FUNCTION_BLOCK LIGHTS_CYCLE (* Composite Function Block Type *)
  (* Standard: 61499-2 *)
  (* Version 0.2, 2003-12-05, JHC, Rockwell Automation, Renamed from NEWCOMPFB. *)
  (* Version 0.1, 2002-01-08, JHC, Rockwell Automation, Added DLY FB as example. *)
  (* Version 0.0, 2000-05-27, JHC, Rockwell Automation *)
  (* Compiler header: package fb.rt.student; *)
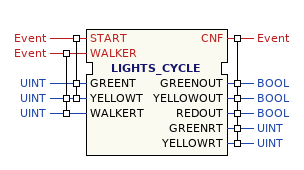
  EVENT_INPUT
    START WITH GREENT, YELLOWT;
    WALKER WITH WALKERT, YELLOWT;
  END_EVENT
  EVENT_OUTPUT
    CNF WITH GREENOUT, YELLOWOUT, REDOUT, GREENRT, YELLOWRT;
  END_EVENT
  VAR_INPUT
    GREENT : UINT;
    YELLOWT : UINT;
    WALKERT : UINT;
  END_VAR
  VAR_OUTPUT
    GREENOUT : BOOL;
    YELLOWOUT : BOOL;
    REDOUT : BOOL;
    GREENRT : UINT;
    YELLOWRT : UINT;
  END_VAR
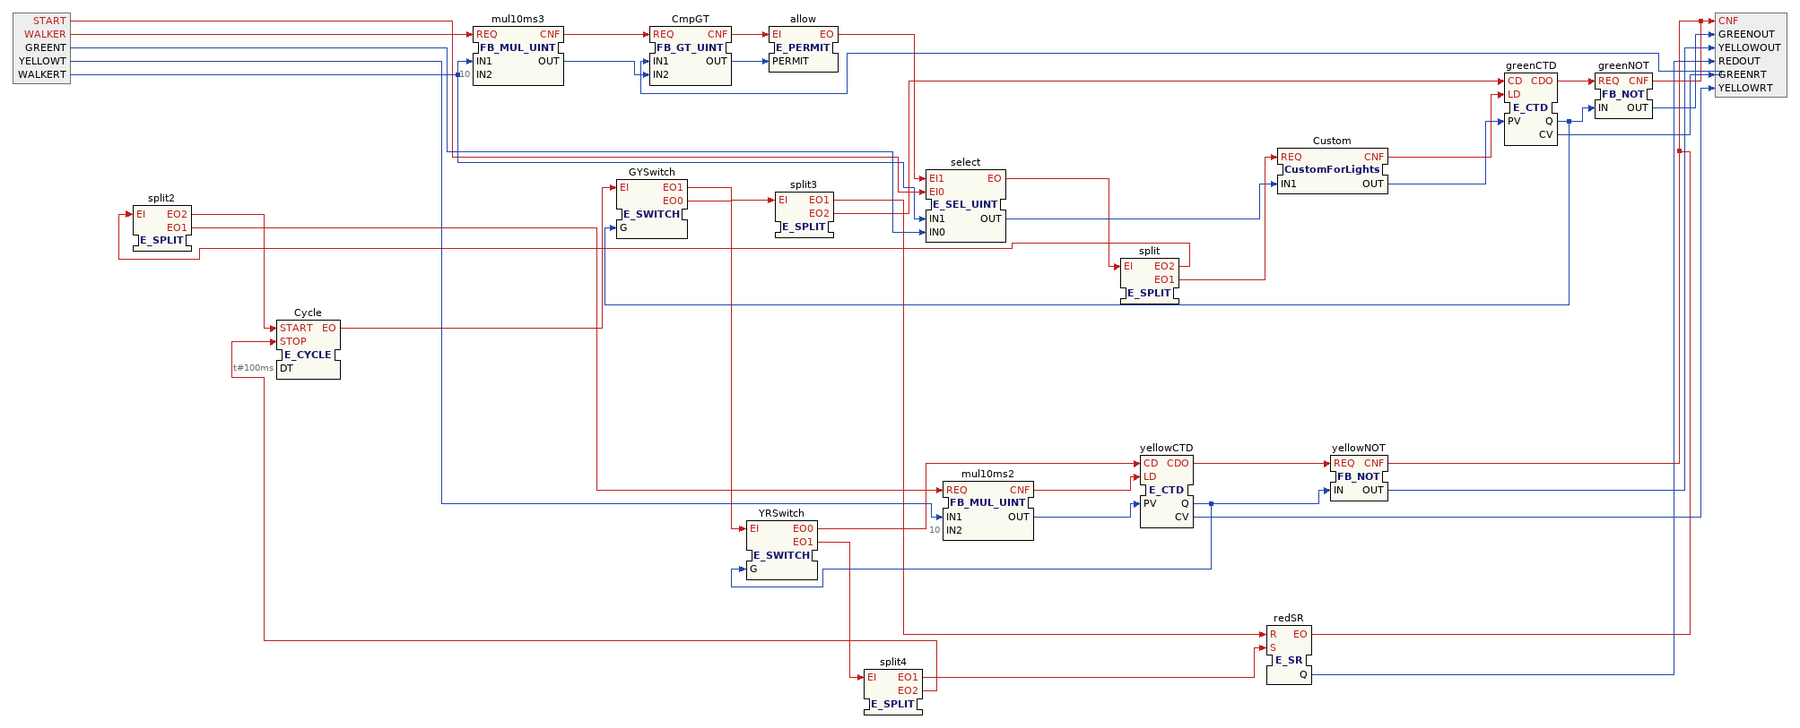
  FBS
    greenCTD : E_CTD;
    yellowCTD : E_CTD;
    Cycle : E_CYCLE(DT := t#100ms);
    GYSwitch : E_SWITCH;
    split : E_SPLIT;
    split2 : E_SPLIT;
    YRSwitch : E_SWITCH;
    redSR : E_SR;
    split3 : E_SPLIT;
    greenNOT : FB_NOT;
    yellowNOT : FB_NOT;
    split4 : E_SPLIT;
    mul10ms2 : FB_MUL_UINT(IN2 := 10);
    CmpGT : FB_GT_UINT;
    allow : E_PERMIT;
    select : E_SEL_UINT;
    mul10ms3 : FB_MUL_UINT(IN2 := 10);
    Custom : CustomForLights;
  END_FBS
  EVENT_CONNECTIONS
    split.EO2 TO split2.EI;
    split2.EO2 TO Cycle.START;
    GYSwitch.EO1 TO YRSwitch.EI;
    YRSwitch.EO0 TO yellowCTD.CD;
    GYSwitch.EO0 TO split3.EI;
    split3.EO1 TO redSR.R;
    split3.EO2 TO greenCTD.CD;
    greenCTD.CDO TO greenNOT.REQ;
    yellowCTD.CDO TO yellowNOT.REQ;
    YRSwitch.EO1 TO split4.EI;
    split4.EO1 TO redSR.S;
    split4.EO2 TO Cycle.STOP;
    split2.EO1 TO mul10ms2.REQ;
    mul10ms2.CNF TO yellowCTD.LD;
    greenNOT.CNF TO CNF;
    yellowNOT.CNF TO CNF;
    redSR.EO TO CNF;
    CmpGT.CNF TO allow.EI;
    allow.EO TO select.EI1;
    START TO select.EI0;
    select.EO TO split.EI;
    mul10ms3.CNF TO CmpGT.REQ;
    WALKER TO mul10ms3.REQ;
    Cycle.EO TO GYSwitch.EI;
    split.EO1 TO Custom.REQ;
    Custom.CNF TO greenCTD.LD;
  END_CONNECTIONS
  DATA_CONNECTIONS
    yellowCTD.Q TO YRSwitch.G;
    redSR.Q TO REDOUT;
    greenCTD.Q TO greenNOT.IN;
    greenNOT.OUT TO GREENOUT;
    yellowCTD.Q TO yellowNOT.IN;
    yellowNOT.OUT TO YELLOWOUT;
    YELLOWT TO mul10ms2.IN1;
    mul10ms2.OUT TO yellowCTD.PV;
    greenCTD.CV TO GREENRT;
    yellowCTD.CV TO YELLOWRT;
    CmpGT.OUT TO allow.PERMIT;
    WALKERT TO select.IN1;
    GREENT TO select.IN0;
    GREENRT TO CmpGT.IN1;
    WALKERT TO mul10ms3.IN1;
    mul10ms3.OUT TO CmpGT.IN2;
    greenCTD.Q TO GYSwitch.G;
    select.OUT TO Custom.IN1;
    Custom.OUT TO greenCTD.PV;
  END_CONNECTIONS
END_FUNCTION_BLOCK
